{attribute 'qualified_only'}
VAR_GLOBAL
	StartOver				: BOOL;
	Stop					: BOOL;
	Pause					: BOOL;
	Resume					: BOOL;
	bzone0Stop				: BOOL;
	SafeToUnlock			: BOOL;
	dsMoverControlFlags		: MoverControlFlags;
	ShuttleMover			: BOOL;
END_VAR

(* stored: Version 1.1.0.1, ProductVersion 3.1.4026.8
   GVL HMI: Id {74764eea-f9f1-0a62-209b-313e6c5f9e7d} *)
